(* PLC project Tc2_Utilities.DCF77_TIME Demo, tc3-libraries-kb TwinCAT 3.1 *)
(* stored: creationDateTime 2026-05-10T20:00:00, modificationDateTime 2026-05-10T20:00:00 *)

PROGRAM P_Demo_DCF77_TIME
  VAR
    fbDCF77_TIME : DCF77_TIME;  (* Tc2_Utilities.DCF77_TIME 实例 *)
    arg_DCF_PULSE : BOOL;  (* VAR_INPUT DCF_PULSE *)
    arg_RUN : BOOL;  (* VAR_INPUT RUN *)
    out_BUSY : BOOL;  (* VAR_OUTPUT BUSY *)
    out_ERR : BOOL;  (* VAR_OUTPUT ERR *)
    out_ERRID : UDINT;  (* VAR_OUTPUT ERRID *)
    out_ERRCNT : UDINT;  (* VAR_OUTPUT ERRCNT *)
    out_READY : BOOL;  (* VAR_OUTPUT READY *)
    out_CDT : DATE_AND_TIME;  (* VAR_OUTPUT CDT *)
  END_VAR

            // ============================================================
// Tc2_Utilities.DCF77_TIME 演示程序（FB 实例）
// ============================================================
// 验证步骤：
//   1. 引用 Tc2_Utilities（及依赖类型所在库 Tc2_System 等）
//   2. 编译 + 登录
//   3. 按 doc.md 给 arg_* 赋值
//   4. 在线监视 out_* / io_* 输出
// ============================================================

fbDCF77_TIME(
    DCF_PULSE := arg_DCF_PULSE,
    RUN := arg_RUN,
    BUSY => out_BUSY,
    ERR => out_ERR,
    ERRID => out_ERRID,
    ERRCNT => out_ERRCNT,
    READY => out_READY,
    CDT => out_CDT
);

          
END_PROGRAM
